{region '#Template'}
	{attribute 'Version' := '1.0.0.0'}
	{attribute 'Tags' := '"LCID": "1031", "Text": "Universal, Control, Ramp limit"'}
	{attribute 'Tags' := '"LCID": "1033", "Text": "Universal, Control, Ramp limit"'}
	{attribute 'Description' := '"LCID": "1031", "Text": "Aufsteigende Rampenbegrenzung"'}
	{attribute 'Description' := '"LCID": "1033", "Text": "Rising ramp limit"'}
{endregion}
FUNCTION_BLOCK FB_BA_RampLimitIncrease EXTENDS FB_BA_View 
VAR_INPUT
	bEn			: BOOL;
	bTrig		: BOOL;
END_VAR
VAR_OUTPUT
	fY			: REAL;
END_VAR
VAR_INPUT CONSTANT
	TiUp		: FB_BA_AV_Op;		 										 
	Y			: FB_BA_AV_Op;	
END_VAR
VAR	
	RampFnct	: FB_BA_RampLmt;
	rtrigSync	: R_TRIG;
END_VAR

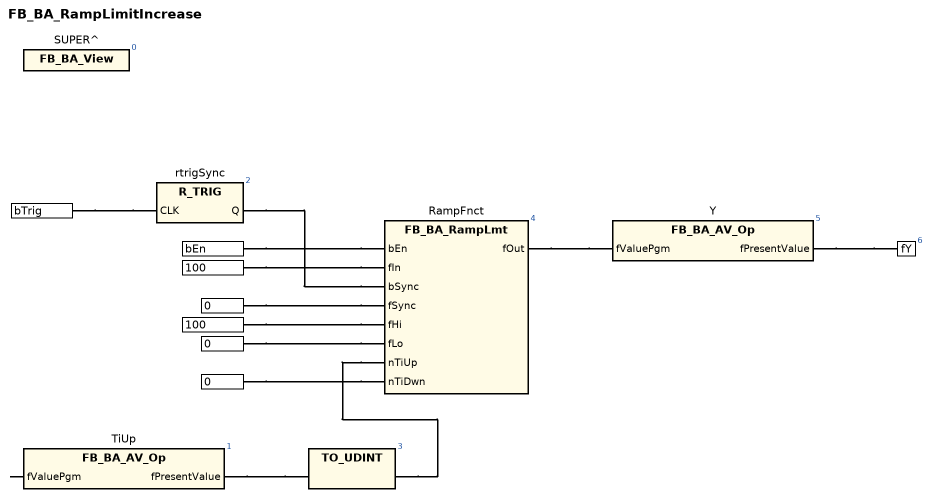
SUPER^(); // FB_BA_View
TiUp(); // FB_BA_AV_Op
rtrigSync(CLK := bTrig); // R_TRIG
RampFnct(
    bEn := bEn,
    fIn := 100,
    bSync := rtrigSync.Q,
    fSync := 0,
    fHi := 100,
    fLo := 0,
    nTiUp := TO_UDINT(TiUp.fPresentValue),
    nTiDwn := 0); // FB_BA_RampLmt
Y(fValuePgm := RampFnct.fOut); // FB_BA_AV_Op
fY := Y.fPresentValue;

METHOD FB_init : BOOL
VAR_INPUT
	bInitRetains : BOOL; // if TRUE, the retain variables are initialized (warm start / cold start)
	bInCopyCode : BOOL;  // if TRUE, the instance afterwards gets moved into the copy code (online change)
END_VAR
TiUp.iParent				:= THIS^;
TiUp.iLabel					:= LblUniControl.Ramp_TiUp;			
TiUp.sObjectName			:= '{Idx=01}';	
TiUp.eUnit					:= E_BA_Unit.eTime_Seconds;								 	 
TiUp.fValueRm				:= 600;
TiUp.fCOVIncrement			:= BA2_Param.fDefCOVIncrement;		

	 										 
Y.iParent					:= THIS^;
Y.iLabel					:= LblUniControl.Ramp_Y;			
Y.sObjectName				:= '{Idx=01}';								 	 
Y.eUnit						:= E_BA_Unit.eOther_Percent;	
Y.fCOVIncrement				:= BA2_Param.fDefCOVIncrement;
END_METHOD

END_FUNCTION_BLOCK

(* stored: Version 1.1.0.1, ProductVersion 3.1.4024.9
   POU FB_BA_RampLimitIncrease: Id {9da2fed4-ed35-4a7b-b03f-dfeebe4b251f}, SpecialFunc None
   Method FB_init: Id {9ac31166-24de-4d2c-b8bc-8a82f2da3a69} *)
